Staubli VAL3: WipeCacheRoom1.pgx

program WipeCacheRoom1()
  local num nNum
begin

  for nNum=0 to 499
    sString[nNum]=""
    pfrmCad[nNum].trsf={0,0,0,0,0,0}
  endFor

end
